Staubli VAL3: convert.pgx

public program convert(joint& x_jJoint, mdesc& x_mMdesc)
  local num l_nRadian2Deg
begin
  // SEQUENCE
  //   END_TRAJECTORY -3
  //   STOP_TRAJECTORY -4
  if body.sequence == -4
    stopMove()
    resetMotion()
  elseIf body.sequence == -3
    x_mMdesc.blend=off
    x_mMdesc.leave=0
    x_mMdesc.reach=0
  else
    x_mMdesc.blend=Cartesian
    // mm
    x_mMdesc.leave=25
    x_mMdesc.reach=25
  endIf

  l_nRadian2Deg = 180 / 3.14159265359

  // POSITION 0x02
  if bAnd(body.validFields,2) == 2
    x_jJoint.j1=body.positions[0] * l_nRadian2Deg
    x_jJoint.j2=body.positions[1] * l_nRadian2Deg
    x_jJoint.j3=body.positions[2] * l_nRadian2Deg
    x_jJoint.j4=body.positions[3] * l_nRadian2Deg
    x_jJoint.j5=body.positions[4] * l_nRadian2Deg
    x_jJoint.j6=body.positions[5] * l_nRadian2Deg
  endIf

  // default values
  x_mMdesc.accel=100
  x_mMdesc.vel=100
  x_mMdesc.decel=100
  x_mMdesc.tvel=99999
  x_mMdesc.rvel=99999

  // VELOCITY 0x04
  if bAnd(body.validFields,4) == 4
    // percent
    x_mMdesc.vel=body.velocities[0]
  endIf

  // ACCELERATION 0x08
  if bAnd(body.validFields,8) == 8
    //percent
    x_mMdesc.accel=body.accelerations[0]
    x_mMdesc.decel=body.accelerations[1]
  endIf
end
